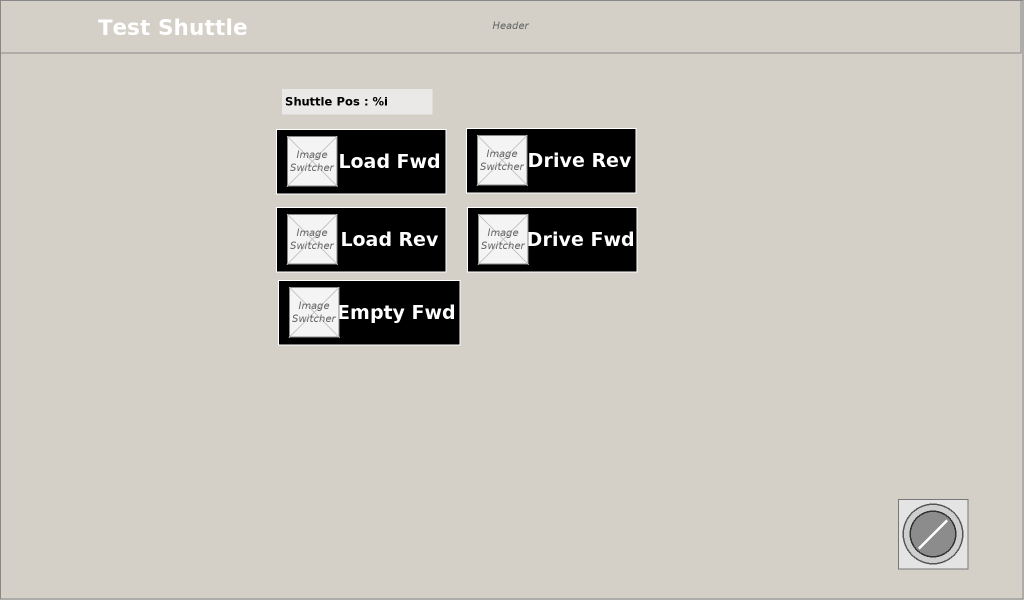
VISUALIZATION Test_Shuttle  // 1024x600
    Frame (0,-2 1021x55)
        shows Header()
    Label (95,15 250x25), "Test Shuttle"
    RotarySwitch (898,499 70x70), variable: HMI_GVL.bTestModeEnableShuttle, behaviour: TOGGLE, style: Switch-RotarySwitch-Gray
    RoundedRectangle (276,129 170x65)
        toggle HMI_GVL.Test_ShuttleLoad_Fwd
    Label (321,149 137x25), "Load Fwd"
    ImageSwitcher (287,136 50x50), variable: HMI_GVL.Test_ShuttleLoad_Fwd, behaviour: TOGGLE
    RoundedRectangle (276,207 170x65)
        toggle HMI_GVL.Test_ShuttleLoad_Rev
    Label (321,227 137x25), "Load Rev"
    ImageSwitcher (287,214 50x50), variable: HMI_GVL.Test_ShuttleLoad_Rev, behaviour: TOGGLE
    RoundedRectangle (278,280 182x65)
        toggle HMI_GVL.Test_ShuttleEmpty_Fwd
    Label (328,300 137x25), "Empty Fwd"
    ImageSwitcher (289,287 50x50), variable: HMI_GVL.Test_ShuttleEmpty_Fwd, behaviour: TOGGLE
    RoundedRectangle (467,207 170x65)
        tap HMI_GVL.Test_ShuttleDrive_Fwd
    Label (512,227 137x25), "Drive Fwd"
    ImageSwitcher (478,214 50x50), variable: HMI_GVL.Test_ShuttleDrive_Fwd, behaviour: TOGGLE
    RoundedRectangle (466,128 170x65)
        tap HMI_GVL.Test_ShuttleDrive_Rev
    Label (511,148 137x25), "Drive Rev"
    ImageSwitcher (477,135 50x50), variable: HMI_GVL.Test_ShuttleDrive_Rev, behaviour: TOGGLE
    Rectangle (282,89 150x25), "Shuttle Pos : %i", text variable: InputOutput_GVL.ShuttlePosition
END_VISUALIZATION

(* stored: Version 1.1.0.1, ProductVersion 3.1.4024.12
   Visu Test_Shuttle: Id {30208145-20f4-47a9-8aa2-4880f6822ff1} *)
